SUBAPPLICATION GreenWhiteBackground_Klappen_senken (* Subapplication Type *)
  (* Standard: 61499-2 *)
  (* Version 1.0, 2023-02-11, franz *)
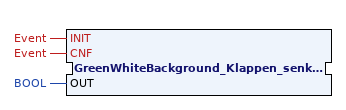
  EVENT_INPUT
    INIT;
    CNF;
  END_EVENT
  VAR_INPUT
    OUT : BOOL;
  END_VAR
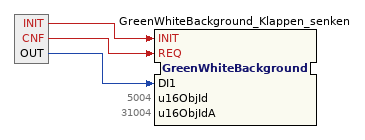
  FBS
    GreenWhiteBackground_Klappen_senken : GreenWhiteBackground(u16ObjId := 5004, u16ObjIdA := 31004);
  END_FBS
  EVENT_CONNECTIONS
    INIT TO GreenWhiteBackground_Klappen_senken.INIT;
    CNF TO GreenWhiteBackground_Klappen_senken.REQ;
  END_CONNECTIONS
  DATA_CONNECTIONS
    OUT TO GreenWhiteBackground_Klappen_senken.DI1;
  END_CONNECTIONS
END_SUBAPPLICATION
